Staubli VAL3: safeCalibration.pjx

--- safeCalibration.pjx ---
Parameters version=s8.5.3Cs9_BS1189 stackSize=5000 millimeterUnit=true
Program file=actBtnFinished.pgx
Program file=start.pgx
Program file=stop.pgx
Program file=tHmi.pgx
Data file=safeCalibration.dtx

--- safeCalibration.dtx ---
bool bEnded
bool bFinished
bool bResult
dio dIrefWarning = {link=Rsi9IO\IrefWarning}
dio dIsafePos = {link=Rsi9IO\IsafePos}
dio dIsafeRec = {link=Rsi9IO\IsafeRec}
dio dIsafeVel = {link=Rsi9IO\IsafeVel}
dio dIwaitingRestart = {link=Rsi9IO\IwaitingRestart}
dio dQrefPos1 = {link=Rsi9IO\QrefPos1}
dio dQrefPos2 = {link=Rsi9IO\QrefPos2}
dio dQresetRef = {link=Rsi9IO\QresetRef}
jointRx jInter[2]
  [0] = {j1=16.747153, j2=23.215229, j3=121.00356449, j4=36.67895, j5=59.788219, j6=-56.84014}
  [1] = {j1=15.334778, j2=29.352505, j3=112.42629, j4=211.510021, j5=-74.522323, j6=-55.937398}
jointRx jSafeReference1 = {j1=-15.981558, j2=6.260298, j3=120.160224, j4=31.4667, j5=66.893497, j6=-29.887624}
jointRx jSafeReference2 = {j1=-3.793248, j2=1.0269555, j3=124.00918551, j4=-180.851639, j5=-30.387886, j6=-41.572914}
jointRx jStart = {j1=-3.793236, j2=0.748011, j3=89.934189, j4=2.918087, j5=83.292851, j6=-41.834364}
jointRx jTmp
jointRx jTolerance = {j1=0.5, j2=0.5, j3=0.5, j4=0.5, j5=0.5, j6=0.5}
mdesc mNomSpeed
num nPrevSafeRefStatus
num nSafeRefStatus
pointRx pTmp = {fatherId=world[0]}
string sBtnFinished
string sHmiBgn{}
  [CurrentStatus] = {}
  [Processing] = {}
  [QrefPos1] = {}
  [QrefPos2] = {}
  [ReqAction] = {}
  [SafePosition] = {}
  [SafeRecovery] = {}
  [SafeVelocity] = {}
string sHmiColor{}
  [CurrentStatus] = {}
  [Processing] = {}
  [QrefPos1] = {}
  [QrefPos2] = {}
  [ReqAction] = {}
  [SafePosition] = {}
  [SafeRecovery] = {}
  [SafeVelocity] = {}
string sHmiColorDef{}
  [DefaultBgn] = {}
  [DefaultColor] = "black"
  [ErrorBgn] = "red"
  [ErrorColor] = "white"
  [InProgressBgn] = "green"
  [InProgressColor] = "black"
  [OffBgn] = "grey"
  [OffColor] = "white"
  [OkBgn] = "lime"
  [OkColor] = "black"
  [OnBgn] = "lime"
  [OnColor] = "black"
  [WarningBgn] = "orange"
  [WarningColor] = "black"
string sHmiStatusBgn{}
  [Checked] = {}
  [Defined] = {}
  [Invalid] = {}
  [Lost] = {}
  [Reset] = {}
  [Warning] = {}
string sHmiStatusColor{}
  [Checked] = {}
  [Defined] = {}
  [Invalid] = {}
  [Lost] = {}
  [Reset] = {}
  [Warning] = {}
string sHmiTxt{}
  [CurrentStatus] = {}
  [Processing] = {}
  [QrefPos1] = {}
  [QrefPos2] = {}
  [ReqAction] = {}
  [SafePosition] = {}
  [SafeRecovery] = {}
  [SafeVelocity] = {}
string sVersion
trsf trAppro
dio dQNoSafePos = {link=Rsi9IO\QnoSafePos}
dio dUSID1 = {link=Rsi9IO\IusiD1}

--- start.pgx ---
program start()
  local bool l_bResult
begin
  // ---------------------------------------------------------------------------------------------
  // Revision history
  //   + means addition
  //   - means removal
  //   ~ means change
  //
  // 20170929 AJAF
  //   + Analysis of safe Velocity, safe Position, safe Recovery status to make only what is needed
  // 20171004 AJAF
  //   + User interface
  // 20171128 AJAF
  //   ~ Conversion to s8.4.1
  //   ~ Hmi task for permanent update.
  // 20180130 AJAF
  //   ~ Correct reset status
  // 20180321 AJAF V5
  //   + Add a disablePower at the start to prevent trouble
  // 20180427 AJAF V6
  //   + Add USID1 activation check
  // ---------------------------------------------------------------------------------------------
  //  jStart: point from which we can start to make safety referencing
  //  jInter[0]: access point to reach first reference point. To be teached
  //  jInter[1]: access point to reach second reference point . To be teached
  //  trAppro: approche done to came close to reference point. to be adjusted below
  // ---------------------------------------------------------------------------------------------


  // Init appro to reference points
  trAppro={0,0,-50,0,0,0}

  // Get safe referencing position
  jSafeReference1=getJntRef("safeReference1")
  jSafeReference2=getJntRef("safeReference2")

  // Init variable
  bFinished=false
  bEnded=true

  taskCreate "tHmi",10,tHmi()
  wait(taskStatus("tHmi")==1)

  // Wait Hmi initialization is finished
  wait(bEnded==false)

  // Display HMI
  userPage("main")

  // Be sure nothing prevent process
  disablePower()
  dioSet(dQNoSafePos,0)

  // Invalid
  if nSafeRefStatus==5
    sHmiTxt["Processing"]="Reference re-initialization ..."
    // Manual mode only
    if workingMode()!=1
      sHmiTxt["ReqAction"]="Waiting manual mode ..."
      wait(workingMode()==1)
      sHmiTxt["ReqAction"]=""
    endIf
    // Reference reinitialization
    dioSet(dQresetRef,0)
    delay(2)
    dioSet(dQresetRef,1)
    delay(2)
    dioSet(dQresetRef,0)
    delay(2)
    // Check if a safety reset is needed
    l_bResult=true
    if (esStatus()==1)
      sHmiTxt["ReqAction"]="Doing safety reset ..."
      l_bResult=setSafetyRestart()
      if l_bResult
        sHmiTxt["ReqAction"]=""
      else
        sHmiTxt["ReqAction"]="Failed to make safety reset."
      endIf
    endIf
  endIf

  // Reset
  if (nSafeRefStatus==4) or (nSafeRefStatus==3)
    sHmiTxt["Processing"]="Doing first reference point ..."
    // Manual mode only
    if workingMode()!=1
      sHmiTxt["ReqAction"]="Waiting manual mode ..."
      wait(workingMode()==1)
      sHmiTxt["ReqAction"]=""
    endIf
    // Check if a safety reset is needed
    l_bResult=true
    if (esStatus()==1)
      sHmiTxt["ReqAction"]="Doing safety reset ..."
      l_bResult=setSafetyRestart()
      if l_bResult
        sHmiTxt["ReqAction"]=""
      else
        sHmiTxt["ReqAction"]="Failed to make safety reset."
      endIf
    endIf
    if l_bResult
      // Arm power ON
      sHmiTxt["ReqAction"]="Please turn arm power ON"
      wait(isPowered())
      sHmiTxt["ReqAction"]=""
      // Go to zero
      resetMotion(jStart)
      // Do first referencing
      movej(jInter[0],flange,mNomSpeed)
      pTmp=appro(jointToPoint(flange,world,jSafeReference1),trAppro)
      bResult=pointToJoint(flange,jSafeReference1,pTmp,jTmp)
      if bResult
        movej(jTmp,flange,mNomSpeed)
      endIf
      movej(jSafeReference1,flange,mNomSpeed)
      waitEndMove()
      disablePower()
      delay(0.5)

      if(herej()!=jSafeReference1) and (dioGet(dQrefPos1)==0)
        sHmiTxt["Processing"]="Warning: At least one axis has moved during first reference point. Check current position compared to safety ones."
        sHmiBgn["Processing"]=sHmiColorDef["WarningBgn"]
      endIf

      if dioGet(dUSID1)==0
        sHmiTxt["Processing"]="Error: USID1 is not activated. Check sensor connected on USID1"
        sHmiColor["Processing"]=sHmiColorDef["ErrorColor"]
        sHmiBgn["Processing"]=sHmiColorDef["ErrorBgn"]
        sHmiTxt["CurrentStatus"]="Sensor on USID1 not working"
      endIf

      if workingMode()==1
        sHmiTxt["ReqAction"]="Please turn arm power ON"
        wait(isPowered())
        sHmiTxt["ReqAction"]=""
      else
        enablePower()
      endIf
      if bResult
        movej(jTmp,flange,mNomSpeed)
      endIf
      movej(jInter[0],flange,mNomSpeed)
      waitEndMove()
    endIf
  endIf

  // Defined or in warning period
  if (nSafeRefStatus==2) or (nSafeRefStatus==1)
    sHmiTxt["Processing"]="Doing second reference point ..."
    // Manual or remote mode only
    if workingMode()!=1 and workingMode()!=4
      sHmiTxt["ReqAction"]="Waiting manual or remote mode ..."
      wait((workingMode()==1) or (workingMode()==4))
      sHmiTxt["ReqAction"]=""
    endIf
    // Check if a safety reset is needed
    l_bResult=true
    if (esStatus()==1)
      sHmiTxt["ReqAction"]="Doing safety reset ..."
      l_bResult=setSafetyRestart()
      if l_bResult
        sHmiTxt["ReqAction"]=""
      else
        sHmiTxt["ReqAction"]="Failed to make safety reset."
      endIf
    endIf
    if l_bResult
      // Arm power ON
      if workingMode()==1
        sHmiTxt["ReqAction"]="Please turn arm power ON"
        wait(isPowered())
        sHmiTxt["ReqAction"]=""
      else
        enablePower()
      endIf
      // Go to jStart if not close to jInter
      if(abs(herej()-jInter[0])>jTolerance) and (abs(herej()-jInter[1])>jTolerance)
        movej(jStart,flange,mNomSpeed)
      endIf
      // Do second referencing
      movej(jInter[1],flange,mNomSpeed)
      pTmp=appro(jointToPoint(flange,world,jSafeReference2),trAppro)
      bResult=pointToJoint(flange,jSafeReference2,pTmp,jTmp)
      if bResult
        movej(jTmp,flange,mNomSpeed)
      endIf
      movej(jSafeReference2,flange,mNomSpeed)
      waitEndMove()
      disablePower()
      delay(0.5)

      if dioGet(dUSID1)==0
        sHmiTxt["Processing"]="Error: USID1 is not activated. Check sensor connected on USID1"
        sHmiColor["Processing"]=sHmiColorDef["ErrorColor"]
        sHmiBgn["Processing"]=sHmiColorDef["ErrorBgn"]
        sHmiTxt["CurrentStatus"]="Sensor on USID1 not working"
      endIf

      if workingMode()==1
        sHmiTxt["ReqAction"]="Please turn arm power ON"
        wait(isPowered())
        sHmiTxt["ReqAction"]=""
      else
        enablePower()
      endIf
      if bResult
        movej(jTmp,flange,mNomSpeed)
      endIf
      movej(jStart,flange,mNomSpeed)
      waitEndMove()
      disablePower()
    endIf
  endIf
  bEnded=true

  // Finished
  wait(bFinished)
end

--- actBtnFinished.pgx ---
program actBtnFinished()
begin
  bFinished=true
end

--- tHmi.pgx ---
program tHmi()
  local string l_sIndex
begin
  // Situation analysis
  // ------------------
  // Safe position OFF, Safe velocity OFF, Safe recovery OFF -> Invalid -> Reinit
  // Safe position OFF, Safe velocity ON, Safe recovery OFF  -> Reset -> Goto refPos1
  // Safe position OFF, Safe velocity OFF, Safe recovery ON  -> Lost -> Goto refPos1
  // Safe position ON, Safe velocity OFF, Safe recovery ON   -> Defined -> Goto refPos2
  // Safe position ON, Safe velocity OFF, Safe recovery OFF  -> Checked

  // Init variables
  sVersion="V6.0"
  l_sIndex=first(sHmiBgn)
  // Background
  while l_sIndex!=""
    sHmiBgn[l_sIndex]=""
    l_sIndex=next(sHmiBgn[l_sIndex])
  endWhile
  // Color
  l_sIndex=first(sHmiColor)
  while l_sIndex!=""
    sHmiColor[l_sIndex]=sHmiColorDef["DefaultColor"]
    l_sIndex=next(sHmiColor[l_sIndex])
  endWhile
  // Text
  l_sIndex=first(sHmiTxt)
  while l_sIndex!=""
    sHmiTxt[l_sIndex]=""
    l_sIndex=next(sHmiTxt[l_sIndex])
  endWhile

  sBtnFinished="hidden"
  nSafeRefStatus=abs(getSafeRefStatus())
  nPrevSafeRefStatus=-2000
  bEnded=false

  while !bEnded
    // QrefPos1
    if dioGet(dQrefPos1)==0
      sHmiTxt["QrefPos1"]="Off"
      sHmiColor["QrefPos1"]=sHmiColorDef["OffColor"]
      sHmiBgn["QrefPos1"]=sHmiColorDef["OffBgn"]
    else
      sHmiTxt["QrefPos1"]="On"
      sHmiColor["QrefPos1"]=sHmiColorDef["OnColor"]
      sHmiBgn["QrefPos1"]=sHmiColorDef["OnBgn"]
    endIf

    // QrefPos2
    if dioGet(dQrefPos2)==0
      sHmiTxt["QrefPos2"]="Off"
      sHmiColor["QrefPos2"]=sHmiColorDef["OffColor"]
      sHmiBgn["QrefPos2"]=sHmiColorDef["OffBgn"]
    else
      sHmiTxt["QrefPos2"]="On"
      sHmiColor["QrefPos2"]=sHmiColorDef["OnColor"]
      sHmiBgn["QrefPos2"]=sHmiColorDef["OnBgn"]
    endIf

    // Safe position
    if dioGet(dIsafePos)==0
      sHmiTxt["SafePosition"]="Off"
      sHmiColor["SafePosition"]=sHmiColorDef["OffColor"]
      sHmiBgn["SafePosition"]=sHmiColorDef["OffBgn"]
    else
      sHmiTxt["SafePosition"]="On"
      sHmiColor["SafePosition"]=sHmiColorDef["OnColor"]
      sHmiBgn["SafePosition"]=sHmiColorDef["OnBgn"]
    endIf

    // Safe velocity
    if dioGet(dIsafeVel)==0
      sHmiTxt["SafeVelocity"]="Off"
      sHmiColor["SafeVelocity"]=sHmiColorDef["OffColor"]
      sHmiBgn["SafeVelocity"]=sHmiColorDef["OffBgn"]
    else
      sHmiTxt["SafeVelocity"]="On"
      sHmiColor["SafeVelocity"]=sHmiColorDef["OnColor"]
      sHmiBgn["SafeVelocity"]=sHmiColorDef["OnBgn"]
    endIf

    // Safe recovery
    if dioGet(dIsafeRec)==0
      sHmiTxt["SafeRecovery"]="Off"
      sHmiColor["SafeRecovery"]=sHmiColorDef["OffColor"]
      sHmiBgn["SafeRecovery"]=sHmiColorDef["OffBgn"]
    else
      sHmiTxt["SafeRecovery"]="On"
      sHmiColor["SafeRecovery"]=sHmiColorDef["OnColor"]
      sHmiBgn["SafeRecovery"]=sHmiColorDef["OnBgn"]
    endIf

    // Referencing status
    nSafeRefStatus=abs(getSafeRefStatus())
    if nSafeRefStatus!=nPrevSafeRefStatus

      sHmiColor["CurrentStatus"]=sHmiColorDef["OkColor"]
      sHmiBgn["CurrentStatus"]=""

      l_sIndex=first(sHmiStatusBgn)
      while l_sIndex!=""
        sHmiStatusBgn[l_sIndex]=sHmiColorDef["DefaultBgn"]
        l_sIndex=next(sHmiStatusBgn[l_sIndex])
      endWhile

      l_sIndex=first(sHmiStatusColor)
      while l_sIndex!=""
        sHmiStatusColor[l_sIndex]=sHmiColorDef["DefaultColor"]
        l_sIndex=next(sHmiStatusColor[l_sIndex])
      endWhile

      switch nSafeRefStatus
        case 0
          sHmiTxt["CurrentStatus"]="Checked"
          sHmiStatusColor["Checked"]=sHmiColorDef["OkColor"]
          sHmiStatusBgn["Checked"]=sHmiColorDef["OkBgn"]
        break

        case 1
          sHmiTxt["CurrentStatus"]="Checked but in the timeout delay"
          sHmiStatusColor["Warning"]=sHmiColorDef["WarningColor"]
          sHmiStatusBgn["Warning"]=sHmiColorDef["WarningBgn"]
        break

        case 2
          sHmiTxt["CurrentStatus"]="Defined"
          sHmiStatusColor["Defined"]=sHmiColorDef["InProgressColor"]
          sHmiStatusBgn["Defined"]=sHmiColorDef["InProgressBgn"]
        break

        case 3
          sHmiTxt["CurrentStatus"]="Lost"
          sHmiStatusColor["Lost"]=sHmiColorDef["ErrorColor"]
          sHmiStatusBgn["Lost"]=sHmiColorDef["ErrorBgn"]
        break

        case 4
          sHmiTxt["CurrentStatus"]="Reset"
          sHmiStatusColor["Reset"]=sHmiColorDef["InProgressColor"]
          sHmiStatusBgn["Reset"]=sHmiColorDef["InProgressBgn"]
        break

        case 5
          sHmiTxt["CurrentStatus"]="Invalid"
          sHmiStatusColor["Invalid"]=sHmiColorDef["ErrorColor"]
          sHmiStatusBgn["Invalid"]=sHmiColorDef["ErrorBgn"]
        break

        case 100
          sHmiTxt["CurrentStatus"]="Failed to read safety configuration"
          sHmiColor["CurrentStatus"]=sHmiColorDef["ErrorColor"]
          sHmiBgn["CurrentStatus"]=sHmiColorDef["ErrorBgn"]
        break

        default
          sHmiTxt["CurrentStatus"]="Unknown"
          sHmiColor["CurrentStatus"]=sHmiColorDef["ErrorColor"]
          sHmiBgn["CurrentStatus"]=sHmiColorDef["ErrorBgn"]
        break
      endSwitch
      nPrevSafeRefStatus=nSafeRefStatus
    endIf

    delay(0)
  endWhile

  // Final status
  if bEnded==true and sBtnFinished!="visible"
    sBtnFinished="visible"
    sHmiTxt["Processing"]=""
    sHmiTxt["ReqAction"]=""
    if nSafeRefStatus==0
      sHmiTxt["Processing"]="Safe referencing OK"
      sHmiColor["Processing"]=sHmiColorDef["OkColor"]
      sHmiBgn["Processing"]=sHmiColorDef["OkBgn"]
    else
      sHmiTxt["Processing"]="Safe referencing failed. Status is: "+sHmiTxt["CurrentStatus"]
      sHmiColor["Processing"]=sHmiColorDef["ErrorColor"]
      sHmiBgn["Processing"]=sHmiColorDef["ErrorBgn"]
    endIf
  endIf
end
